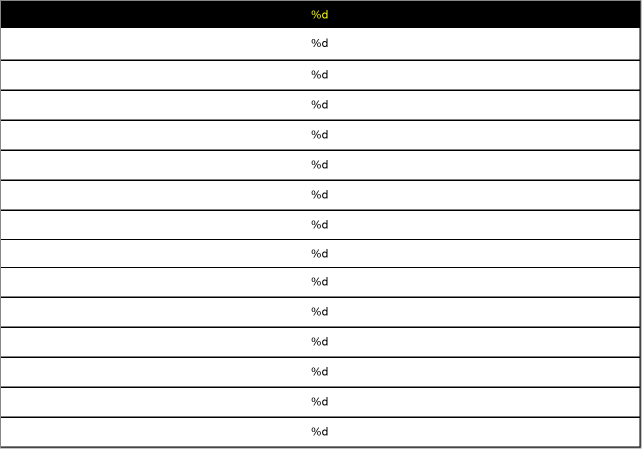
VISUALIZATION CUPS_FEEDING_SHIFT_ELEMENT  // 642x449
VAR_INPUT
	index:		UDINT;
END_VAR
    Rectangle (0,0 640x30), "%d", text variable: csp_case_main_statistics_debug.outer_shift_debug[index].step_id
    Rectangle (0,27 640x33), "%d", text variable: csp_case_main_statistics_debug.outer_shift_debug[index].status.1, colour toggle: csp_case_main_statistics_debug.outer_shift_debug[index].status.1
    Rectangle (0,150 640x30), "%d", text variable: csp_case_main_statistics_debug.outer_shift_debug[index].status.5, colour toggle: csp_case_main_statistics_debug.outer_shift_debug[index].status.5
    Rectangle (0,60 640x30), "%d", text variable: csp_case_main_statistics_debug.outer_shift_debug[index].reject_reason, colour toggle: csp_case_main_statistics_debug.outer_shift_debug[index].reject_reason
    Rectangle (0,180 640x30), "%d", text variable: csp_case_main_statistics_debug.outer_shift_debug[index].status.6, colour toggle: csp_case_main_statistics_debug.outer_shift_debug[index].status.6
    Rectangle (0,120 640x30), "%d", text variable: csp_case_main_statistics_debug.outer_shift_debug[index].status.4, colour toggle: csp_case_main_statistics_debug.outer_shift_debug[index].status.4
    Rectangle (0,210 640x30), "%d", text variable: csp_case_main_statistics_debug.outer_shift_debug[index].status.7, colour toggle: csp_case_main_statistics_debug.outer_shift_debug[index].status.7
    Rectangle (0,239 640x30), "%d", text variable: csp_case_main_statistics_debug.outer_shift_debug[index].status.8, colour toggle: csp_case_main_statistics_debug.outer_shift_debug[index].status.8
    Rectangle (0,267 640x30), "%d", text variable: csp_case_main_statistics_debug.outer_shift_debug[index].status.10, colour toggle: csp_case_main_statistics_debug.outer_shift_debug[index].status.10
    Rectangle (0,297 640x30), "%d", text variable: csp_case_main_statistics_debug.outer_shift_debug[index].status.11, colour toggle: csp_case_main_statistics_debug.outer_shift_debug[index].status.11
    Rectangle (0,327 640x30), "%d", text variable: csp_case_main_statistics_debug.outer_shift_debug[index].status.12, colour toggle: csp_case_main_statistics_debug.outer_shift_debug[index].status.12
    Rectangle (0,357 640x30), "%d", text variable: csp_case_main_statistics_debug.outer_shift_debug[index].status.13, colour toggle: csp_case_main_statistics_debug.outer_shift_debug[index].status.13
    Rectangle (0,387 640x30), "%d", text variable: csp_case_main_statistics_debug.outer_shift_debug[index].status.15, colour toggle: csp_case_main_statistics_debug.outer_shift_debug[index].status.15
    Rectangle (0,417 640x30), "%d", text variable: csp_transfer_main_statistics_debug.transfer_shift_debug[index].status.16, colour toggle: csp_transfer_main_statistics_debug.transfer_shift_debug[index].status.16
    Rectangle (0,90 640x30), "%d", text variable: csp_case_main_statistics_debug.outer_shift_debug[index].status.3, colour toggle: csp_case_main_statistics_debug.outer_shift_debug[index].status.3
END_VISUALIZATION

(* stored: Version 1.1.0.1, ProductVersion 3.1.4024.3
   Visu CUPS_FEEDING_SHIFT_ELEMENT: Id {1a131cf9-3cbe-4010-89c2-26f1a52411bc} *)
